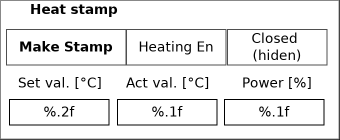
VISUALIZATION vHP3_HeatedStampMain  // 340x140
VAR_IN_OUT
	fbHP	: fbHPv3_Control;
END_VAR
    RoundedRectangle (0,0 340x140), "Heat stamp"
    Rectangle (9,99 100x26), "%.2f", text variable: fbHP.fbHS_PID.SET_POINT
    Label (10,70 100x26), "Set val. [°C]"
    Rectangle (117,99 100x26), "%.1f", text variable: fbHP.fbHS_PID.ACTUAL
    Label (118,70 100x26), "Act val. [°C]"
    Rectangle (224,99 100x26), "%.1f", text variable: fbHP.rHSHeaterPower, colour toggle: fbHP.rHSHeaterPower > 90.0
    Label (225,70 104x26), "Power [%]"
    Rectangle (126,29 100x36), "Heating En", colour toggle: fbHP.fbHS_HeaterON.Q
    Rectangle (227,29 100x36), "Closed (hiden)", colour toggle: fbHP.stInOuts.bI_HeatStampPistonBasePos
    Rectangle (6,29 120x36), "Make Stamp", colour toggle: fbHP.bMakeStamp, input disabled if: NOT fbHP.bMarkingAsembled
        toggle fbHP.bMakeStamp
END_VISUALIZATION

(* stored: Version 1.1.0.1, ProductVersion 3.1.4024.13
   Visu vHP3_HeatedStampMain: Id {75133612-5d9b-4578-be03-cd24488f4780} *)
